(* Logix 5000 project; controller Drives_Line1 1756-L72 rev 20.13; software revision 20.04; part 3 of 21 *)
(* tags used below, declared in another part *)
   Entry_PosPv_Shear_Stitch : REAL;
   Entry_PosPv_Stitch_HOC : DINT;
   Entry_PosSp_AtStitch_EOC : DINT;
   Entry_PosSp_AtStitch_HOC : DINT;
   EOC_PosStitchStep : DINT;
   HOC_ToStitchStep : DINT;
   ons : BOOL[32];
   zEntry_Dist_Pinch_Shear : REAL;
   zEntry_Dist_ShearToStitch : REAL;
   zMaxSpdEntryNotSync : REAL;
   Bridle_01 : UDT_Bridle_3M;
   Bridle_01_FB_Diff : REAL;
   Bridle_01_FB_Update_Valid : BOOL;
   Bridle_01b_FBCounts_mm : REAL;
   Bridle_04 : UDT_Bridle_3M;
   Entry_Accu : UDT_Entry_Accu;
   EntryCmd : UDT_Commands_Zone;
   EntryConfig : UDT_Config_Zone;
   EntryCtrl : UDT_Control_Zone;
   EntryFdbks : UDT_Feedbacks_Zone;
   EntrySetpoints : UDT_Setpoints_Zone;
   EntryStat : UDT_Status_Zone;
   Exit_Accu : UDT_Exit_Accu;
   ExitCmd : UDT_Commands_Zone;
   ExitConfig : UDT_Config_Zone;
   ExitFdbks : UDT_Feedbacks_Zone;
   ExitSetpoints : UDT_Setpoints_Zone;
   ExitStat : UDT_Status_Zone;
   In_Commands : UDT_Commands;
   In_Config : UDT_Config;
   In_Setpoints : UDT_Setpoints;
   LineStat : UDT_Status_Line;
   Out_Feedbacks : UDT_Fdbks;
   Out_Status : UDT_Status;
   Pinchroll_2_FB_Difference : DINT;
   Pinchroll_2_FB_Update_Valid : BOOL;
   Pinchroll_2_FBCounts_mm : REAL;
   Pinchroll_3 : UDT_Pinchroll;
   TestConfig_Entry : UDT_Config_Zone;
   Unwinder_1 : UDT_Unwinder;
   Unwinder_2 : UDT_Unwinder;
   Winder : UDT_Winder;
   zConfigFromMaster : BOOL;
(* P01_Entry_Zone, continued *)

ROUTINE R04a_EOC_ToStitch   (* ladder *)
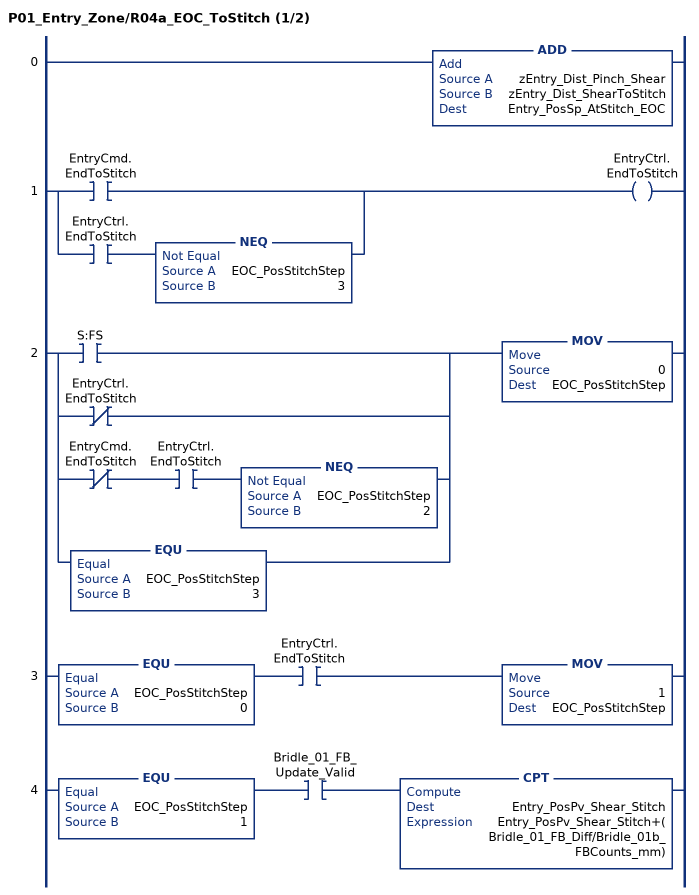
   0: ADD(zEntry_Dist_Pinch_Shear,zEntry_Dist_ShearToStitch,Entry_PosSp_AtStitch_EOC);
   1: [XIC(EntryCmd.EndToStitch) ,XIC(EntryCtrl.EndToStitch) NEQ(EOC_PosStitchStep,3) ]OTE(EntryCtrl.EndToStitch);
   2: [XIC(S:FS) ,XIO(EntryCtrl.EndToStitch) ,XIO(EntryCmd.EndToStitch) XIC(EntryCtrl.EndToStitch) NEQ(EOC_PosStitchStep,2) ,EQU(EOC_PosStitchStep,3) ]MOV(0,EOC_PosStitchStep);
   3: EQU(EOC_PosStitchStep,0)XIC(EntryCtrl.EndToStitch)MOV(1,EOC_PosStitchStep);
   4: EQU(EOC_PosStitchStep,1)XIC(Bridle_01_FB_Update_Valid)CPT(Entry_PosPv_Shear_Stitch,Entry_PosPv_Shear_Stitch+(Bridle_01_FB_Diff/Bridle_01b_FBCounts_mm));
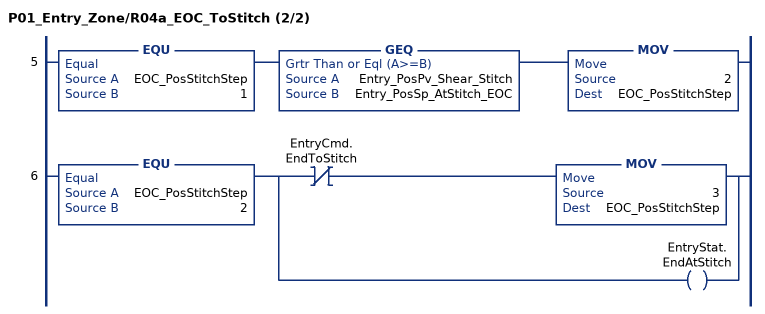
   5: EQU(EOC_PosStitchStep,1)GEQ(Entry_PosPv_Shear_Stitch,Entry_PosSp_AtStitch_EOC)MOV(2,EOC_PosStitchStep);
   6: EQU(EOC_PosStitchStep,2)[XIO(EntryCmd.EndToStitch) MOV(3,EOC_PosStitchStep) ,OTE(EntryStat.EndAtStitch) ];
END_ROUTINE

ROUTINE R04b_HOC_ToStitch   (* ladder *)
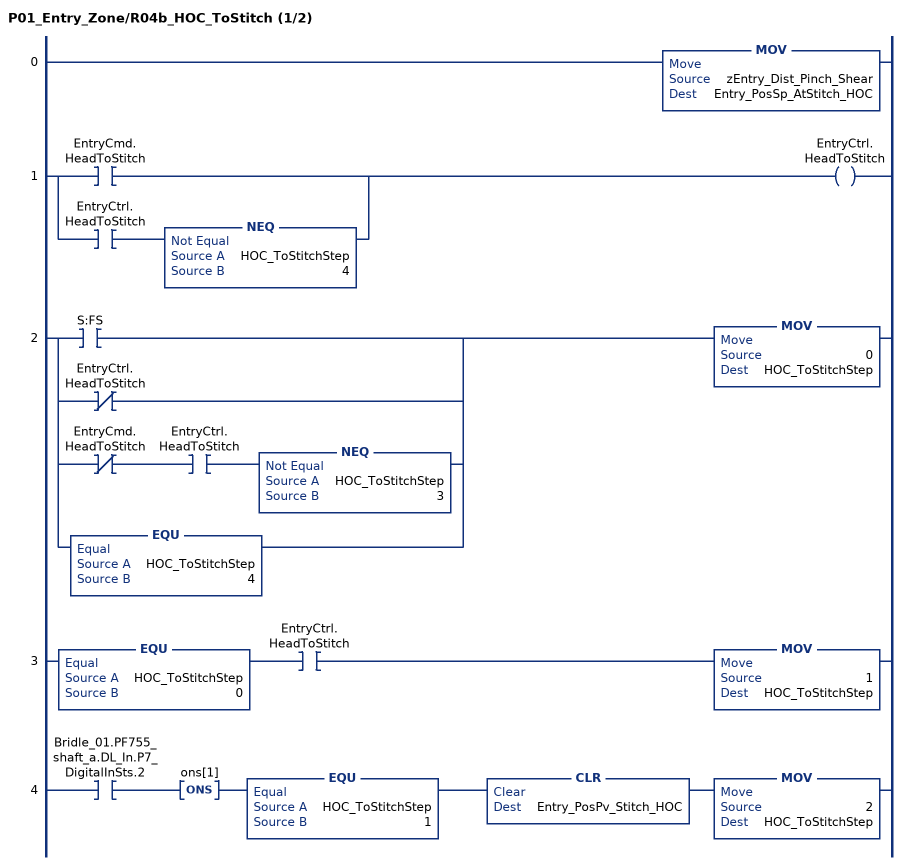
   0: MOV(zEntry_Dist_Pinch_Shear,Entry_PosSp_AtStitch_HOC);
   1: [XIC(EntryCmd.HeadToStitch) ,XIC(EntryCtrl.HeadToStitch) NEQ(HOC_ToStitchStep,4) ]OTE(EntryCtrl.HeadToStitch);
   2: [XIC(S:FS) ,XIO(EntryCtrl.HeadToStitch) ,XIO(EntryCmd.HeadToStitch) XIC(EntryCtrl.HeadToStitch) NEQ(HOC_ToStitchStep,3) ,EQU(HOC_ToStitchStep,4) ]MOV(0,HOC_ToStitchStep);
   3: EQU(HOC_ToStitchStep,0)XIC(EntryCtrl.HeadToStitch)MOV(1,HOC_ToStitchStep);
   4: XIC(Bridle_01.PF755_shaft_a.DL_In.P7_DigitalInSts.2)ONS(ons[1])EQU(HOC_ToStitchStep,1)CLR(Entry_PosPv_Stitch_HOC)MOV(2,HOC_ToStitchStep);
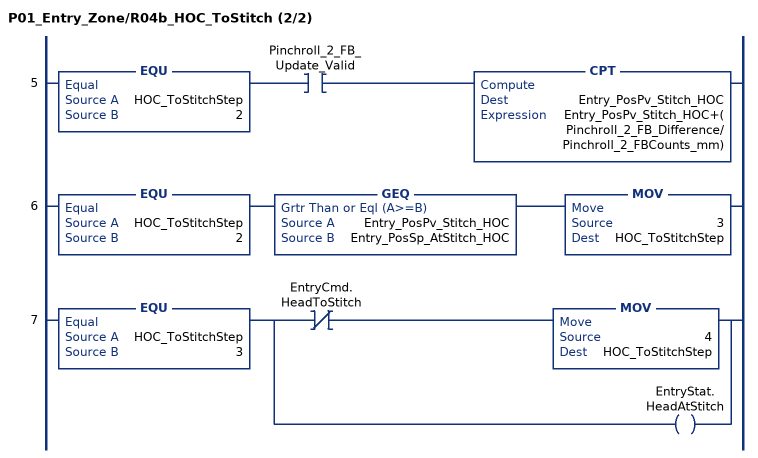
   5: EQU(HOC_ToStitchStep,2)XIC(Pinchroll_2_FB_Update_Valid)CPT(Entry_PosPv_Stitch_HOC,Entry_PosPv_Stitch_HOC+(Pinchroll_2_FB_Difference/Pinchroll_2_FBCounts_mm));
   6: EQU(HOC_ToStitchStep,2)GEQ(Entry_PosPv_Stitch_HOC,Entry_PosSp_AtStitch_HOC)MOV(3,HOC_ToStitchStep);
   7: EQU(HOC_ToStitchStep,3)[XIO(EntryCmd.HeadToStitch) MOV(4,HOC_ToStitchStep) ,OTE(EntryStat.HeadAtStitch) ];
END_ROUTINE

ROUTINE R06_Control   (* ladder *)
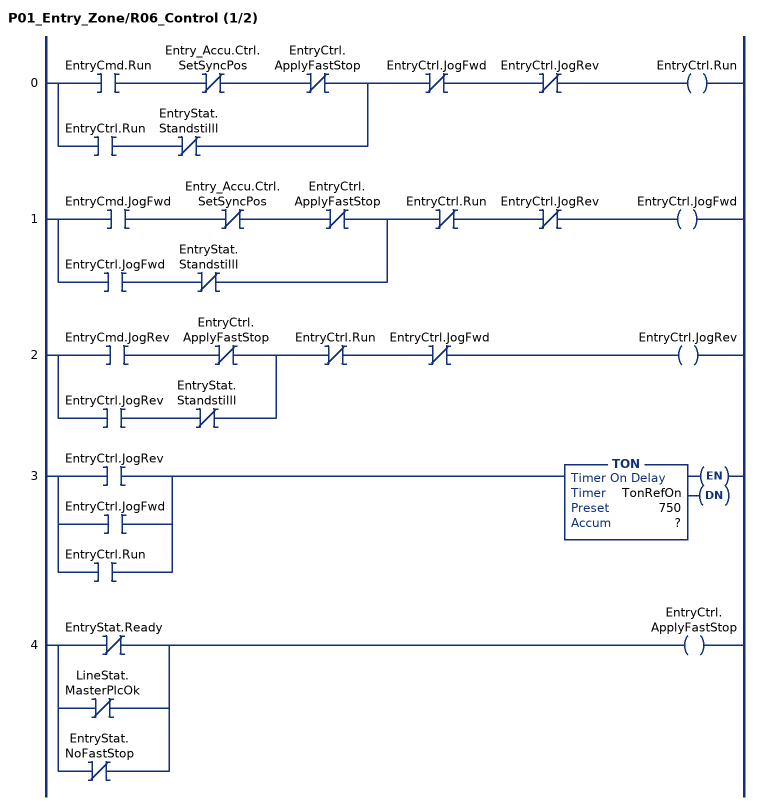
   0: [XIC(EntryCmd.Run) XIO(Entry_Accu.Ctrl.SetSyncPos) XIO(EntryCtrl.ApplyFastStop) ,XIC(EntryCtrl.Run) XIO(EntryStat.Standstilll) ]XIO(EntryCtrl.JogFwd)XIO(EntryCtrl.JogRev)OTE(EntryCtrl.Run);
   1: [XIC(EntryCmd.JogFwd) XIO(Entry_Accu.Ctrl.SetSyncPos) XIO(EntryCtrl.ApplyFastStop) ,XIC(EntryCtrl.JogFwd) XIO(EntryStat.Standstilll) ]XIO(EntryCtrl.Run)XIO(EntryCtrl.JogRev)OTE(EntryCtrl.JogFwd);
   2: [XIC(EntryCmd.JogRev) XIO(EntryCtrl.ApplyFastStop) ,XIC(EntryCtrl.JogRev) XIO(EntryStat.Standstilll) ]XIO(EntryCtrl.Run)XIO(EntryCtrl.JogFwd)OTE(EntryCtrl.JogRev);
   3: [XIC(EntryCtrl.JogRev) ,XIC(EntryCtrl.JogFwd) ,XIC(EntryCtrl.Run) ]TON(TonRefOn,?,?);
   4: [XIO(EntryStat.Ready) ,XIO(LineStat.MasterPlcOk) ,XIO(EntryStat.NoFastStop) ]OTE(EntryCtrl.ApplyFastStop);
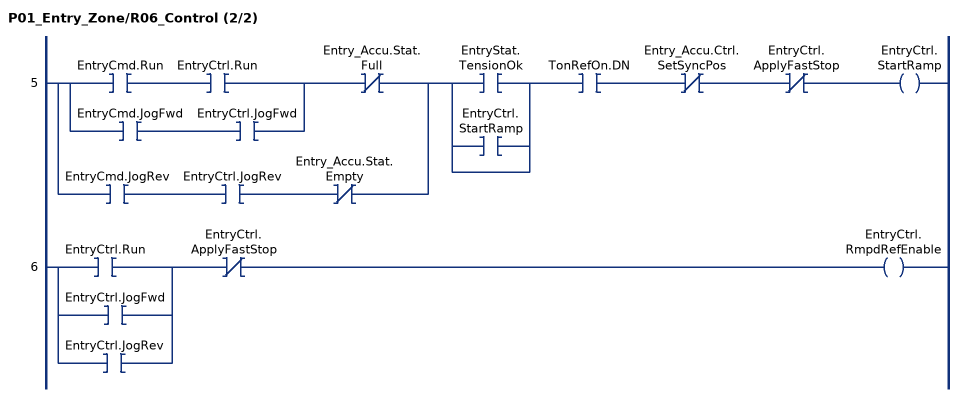
   5: [[XIC(EntryCmd.Run) XIC(EntryCtrl.Run) ,XIC(EntryCmd.JogFwd) XIC(EntryCtrl.JogFwd) ] XIO(Entry_Accu.Stat.Full) ,XIC(EntryCmd.JogRev) XIC(EntryCtrl.JogRev) XIO(Entry_Accu.Stat.Empty) ][XIC(EntryStat.TensionOk) ,XIC(EntryCtrl.StartRamp) ,]XIC(TonRefOn.DN)XIO(Entry_Accu.Ctrl.SetSyncPos)XIO(EntryCtrl.ApplyFastStop)OTE(EntryCtrl.StartRamp);
   6: [XIC(EntryCtrl.Run) ,XIC(EntryCtrl.JogFwd) ,XIC(EntryCtrl.JogRev) ]XIO(EntryCtrl.ApplyFastStop)OTE(EntryCtrl.RmpdRefEnable);
END_ROUTINE

ROUTINE R07_Ramp_EntryRef_Ve   (* function block diagram *)
   SHEET 1   // Limit speed reference
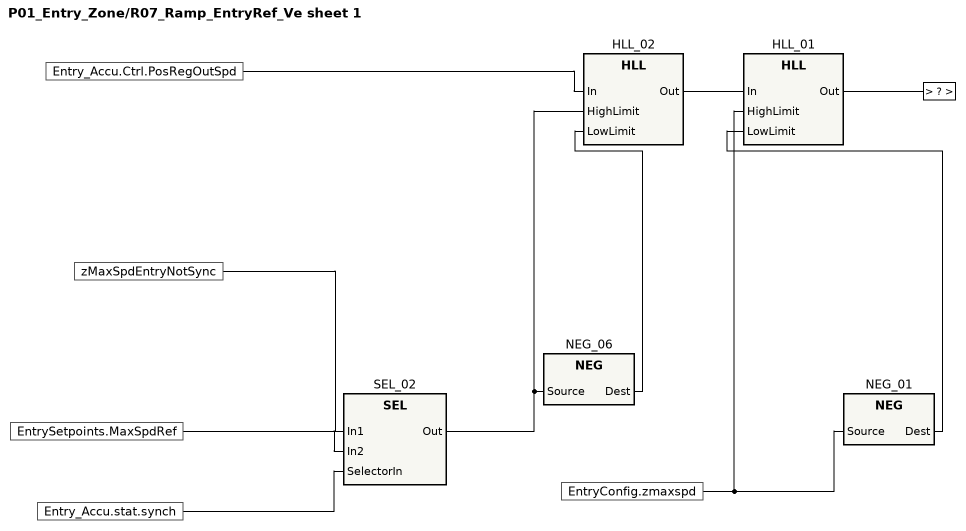
   SEL_02 : SEL(In1 := zMaxSpdEntryNotSync, In2 := EntrySetpoints.MaxSpdRef, SelectorIn := Entry_Accu.stat.synch);
   NEG_06 : NEG(Source := SEL_02.Out);
   HLL_02 : HLL(In := Entry_Accu.Ctrl.PosRegOutSpd, HighLimit := SEL_02.Out, LowLimit := NEG_06.Dest);
   NEG_01 : NEG(Source := EntryConfig.zmaxspd);
   HLL_01 : HLL(In := HLL_02.Out, HighLimit := EntryConfig.zmaxspd, LowLimit := NEG_01.Dest);
   WIRE(?) := HLL_01.Out;
   SHEET 2   // Select reference
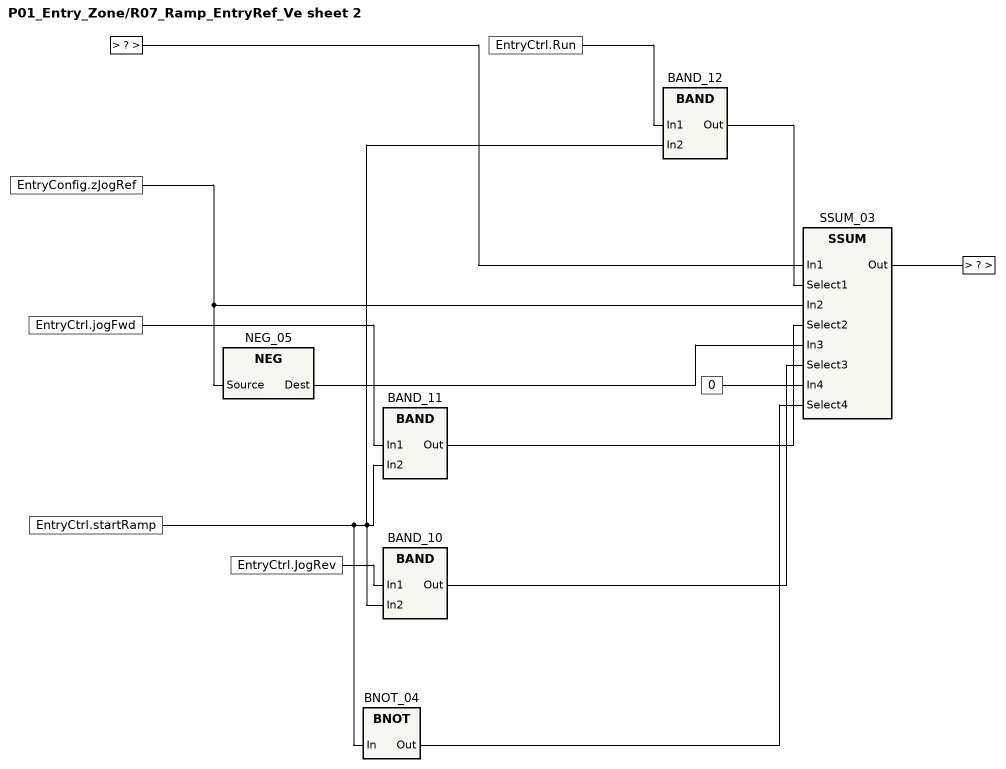
   NEG_05 : NEG(Source := EntryConfig.zJogRef);
   BNOT_04 : BNOT(In := EntryCtrl.startRamp);
   BAND_11 : BAND(In1 := EntryCtrl.jogFwd, In2 := EntryCtrl.startRamp);
   BAND_10 : BAND(In1 := EntryCtrl.JogRev, In2 := EntryCtrl.startRamp);
   BAND_12 : BAND(In1 := EntryCtrl.Run, In2 := EntryCtrl.startRamp);
   SSUM_03 : SSUM(In1 := WIRE(?), Select1 := BAND_12.Out, In2 := EntryConfig.zJogRef, Select2 := BAND_11.Out, In3 := NEG_05.Dest, Select3 := BAND_10.Out, In4 := 0, Select4 := BNOT_04.Out);
   WIRE(?) := SSUM_03.Out;
   SHEET 3   // Select acceleration rate
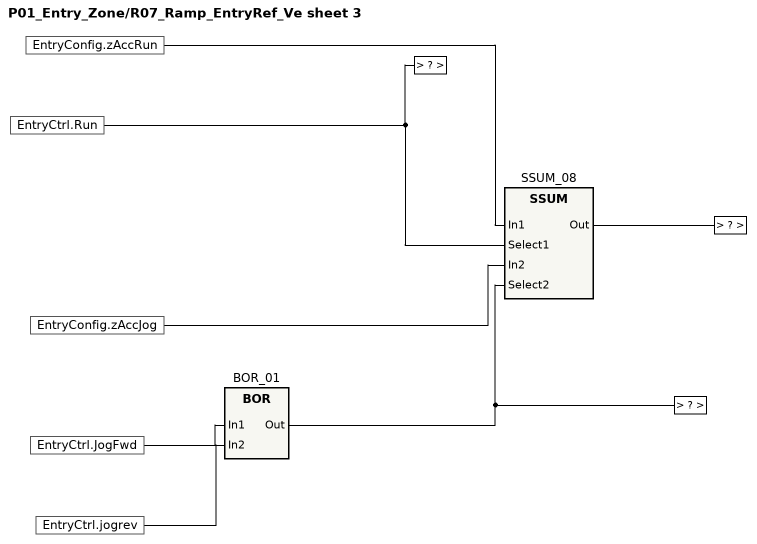
   BOR_01 : BOR(In1 := EntryCtrl.JogFwd, In2 := EntryCtrl.jogrev);
   WIRE(?) := EntryCtrl.Run;
   SSUM_08 : SSUM(In1 := EntryConfig.zAccRun, Select1 := EntryCtrl.Run, In2 := EntryConfig.zAccJog, Select2 := BOR_01.Out);
   WIRE(?) := BOR_01.Out;
   WIRE(?) := SSUM_08.Out;
   SHEET 4   // Select deceleration rate
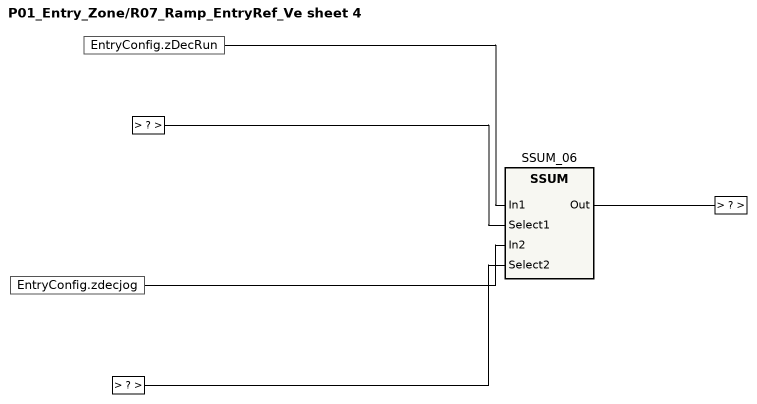
   SSUM_06 : SSUM(In1 := EntryConfig.zDecRun, Select1 := WIRE(?), In2 := EntryConfig.zdecjog, Select2 := WIRE(?));
   WIRE(?) := SSUM_06.Out;
   SHEET 5   // Select jerk rate
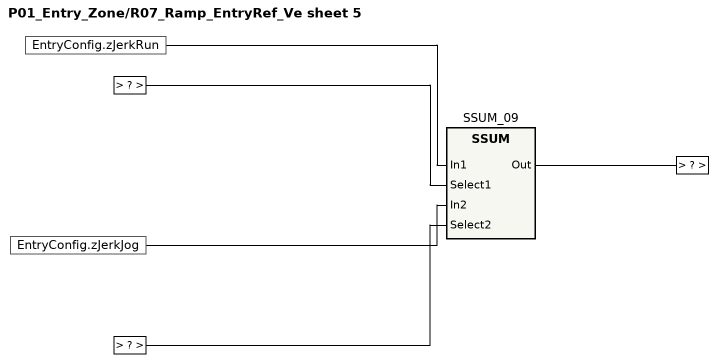
   SSUM_09 : SSUM(In1 := EntryConfig.zJerkRun, Select1 := WIRE(?), In2 := EntryConfig.zJerkJog, Select2 := WIRE(?));
   WIRE(?) := SSUM_09.Out;
   SHEET 6   // S-Curve entry speed (Ve)
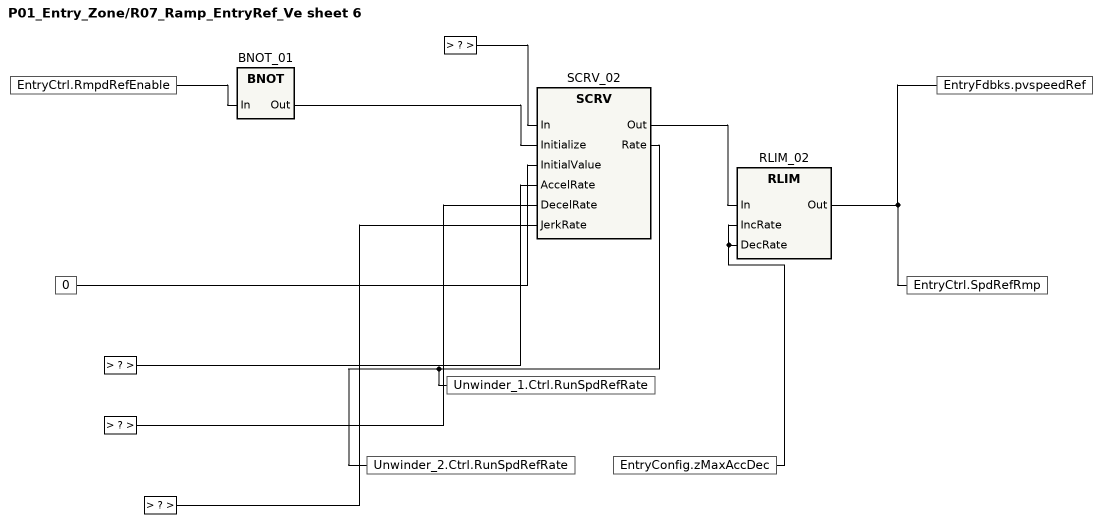
   BNOT_01 : BNOT(In := EntryCtrl.RmpdRefEnable);
   SCRV_02 : SCRV(In := WIRE(?), Initialize := BNOT_01.Out, InitialValue := 0, AccelRate := WIRE(?), DecelRate := WIRE(?), JerkRate := WIRE(?));
   Unwinder_2.Ctrl.RunSpdRefRate := SCRV_02.Rate;
   Unwinder_1.Ctrl.RunSpdRefRate := SCRV_02.Rate;
   RLIM_02 : RLIM(In := SCRV_02.Out, IncRate := EntryConfig.zMaxAccDec, DecRate := EntryConfig.zMaxAccDec);
   EntryCtrl.SpdRefRmp := RLIM_02.Out;
   EntryFdbks.pvspeedRef := RLIM_02.Out;
END_ROUTINE

ROUTINE R999_Test   (* ladder *)
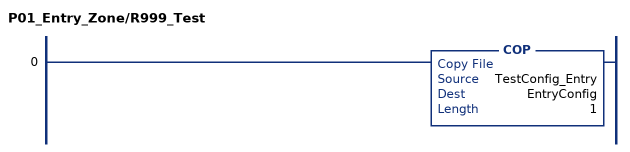
   0: COP(TestConfig_Entry,EntryConfig,1);
END_ROUTINE

ROUTINE R99_To_Master   (* ladder *)
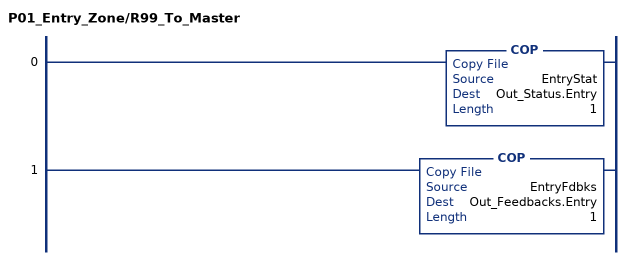
   0: COP(EntryStat,Out_Status.Entry,1);
   1: COP(EntryFdbks,Out_Feedbacks.Entry,1);
END_ROUTINE
END_PROGRAM

PROGRAM P02_Exit_Zone   (* main routine R00_Main *)
VAR
   BAND_10 : FBD_BOOLEAN_AND := (In3 := 1, In4 := 1, In5 := 1, In6 := 1, In7 := 1, In8 := 1);
   BAND_11 : FBD_BOOLEAN_AND := (In3 := 1, In4 := 1, In5 := 1, In6 := 1, In7 := 1, In8 := 1);
   BAND_12 : FBD_BOOLEAN_AND := (In3 := 1, In4 := 1, In5 := 1, In6 := 1, In7 := 1, In8 := 1);
   BNOT_02 : FBD_BOOLEAN_NOT := (Out := 1);
   BNOT_04 : FBD_BOOLEAN_NOT := (Out := 1);
   BOR_02 : FBD_BOOLEAN_OR;
   DIV_02 : FBD_MATH := (SourceA := 70.46141, SourceB := 100.0, Dest := 0.7046141);
   EOC_ToCoilerStep : DINT;
   Exit_PosPv_Winder : REAL;
   HLL_03 : HL_LIMIT := (HighAlarm := 1, LowAlarm := 1, Status := 16#0000_0003, InstructFault := 1, LimitsInv := 1);
   HLL_04 : HL_LIMIT := (HighLimit := 0.35230705, LowLimit := -0.35230705);
   MUL_02 : FBD_MATH := (SourceA := 0.5, SourceB := 0.7046141, Dest := 0.35230705);
   NEG_04 : FBD_MATH_ADVANCED := (Source := 0.35230705, Dest := -0.35230705);
   NEG_05 : FBD_MATH_ADVANCED := (Source := 0.116, Dest := -0.116);
   NEG_06 : FBD_MATH_ADVANCED;
   RLIM_03 : RATE_LIMITER := (IncRate := 0.25, DecRate := 0.25, RTSTime := 1, DeltaT := 0.05);
   SCL_02 : SCALE := (In := 709.3403, InRawMax := 1000.0, InRawMin := 508.0, InEUMax := 100.0, InEUMin := 50.0, Limiting := 1, Out := 70.46141);
   SCRV_03 : S_CURVE := (Initialize := 1, RTSTime := 1, DeltaT := 0.05);
   SEL_02 : SELECT := (In1 := 0.025, SelectorIn := 1);
   SSUM_03 : SELECTED_SUMMER := (Gain1 := 1.0, In2 := 0.116, Gain2 := 1.0, In3 := -0.116, Gain3 := 1.0, Gain4 := 1.0, Select4 := 1, Gain5 := 1.0, Gain6 := 1.0, Gain7 := 1.0, Gain8 := 1.0);
   SSUM_07 : SELECTED_SUMMER := (In1 := 0.04, Gain1 := 1.0, In2 := 0.083, Gain2 := 1.0, Gain3 := 1.0, Gain4 := 1.0, Gain5 := 1.0, Gain6 := 1.0, Gain7 := 1.0, Gain8 := 1.0);
   SSUM_10 : SELECTED_SUMMER := (In1 := 0.04, Gain1 := 1.0, In2 := 0.083, Gain2 := 1.0, Gain3 := 1.0, Gain4 := 1.0, Gain5 := 1.0, Gain6 := 1.0, Gain7 := 1.0, Gain8 := 1.0);
   SSUM_11 : SELECTED_SUMMER := (In1 := 0.15, Gain1 := 1.0, In2 := 0.25, Gain2 := 1.0, Gain3 := 1.0, Gain4 := 1.0, Gain5 := 1.0, Gain6 := 1.0, Gain7 := 1.0, Gain8 := 1.0);
   TonRefOn : TIMER := (PRE := 750);
   zMaxSpdExitNotSync : REAL := 0.025;
END_VAR

ROUTINE R00_Main   (* ladder *)
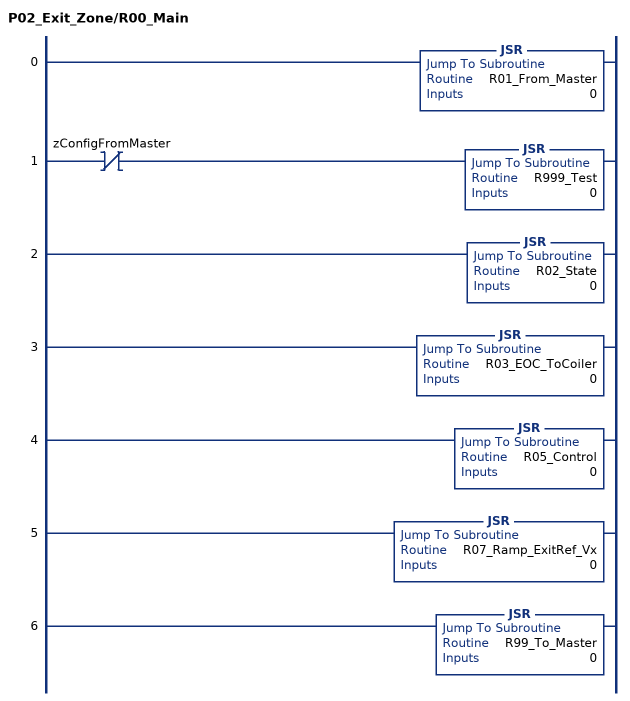
   0: JSR(R01_From_Master,0);
   1: XIO(zConfigFromMaster)JSR(R999_Test,0);
   2: JSR(R02_State,0);
   3: JSR(R03_EOC_ToCoiler,0);
   4: JSR(R05_Control,0);
   5: JSR(R07_Ramp_ExitRef_Vx,0);
   6: JSR(R99_To_Master,0);
END_ROUTINE

ROUTINE R01_From_Master   (* ladder *)
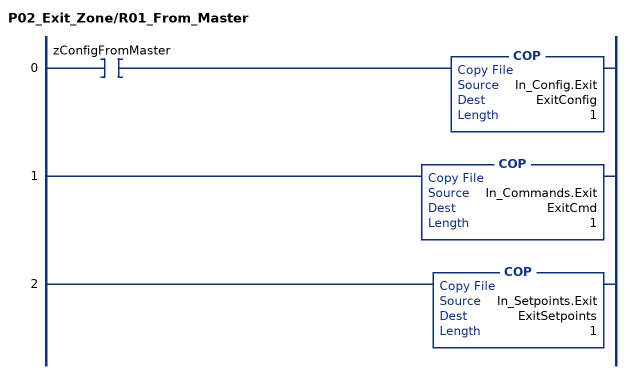
   0: XIC(zConfigFromMaster)COP(In_Config.Exit,ExitConfig,1);
   1: COP(In_Commands.Exit,ExitCmd,1);
   2: COP(In_Setpoints.Exit,ExitSetpoints,1);
END_ROUTINE

ROUTINE R02_State   (* ladder *)
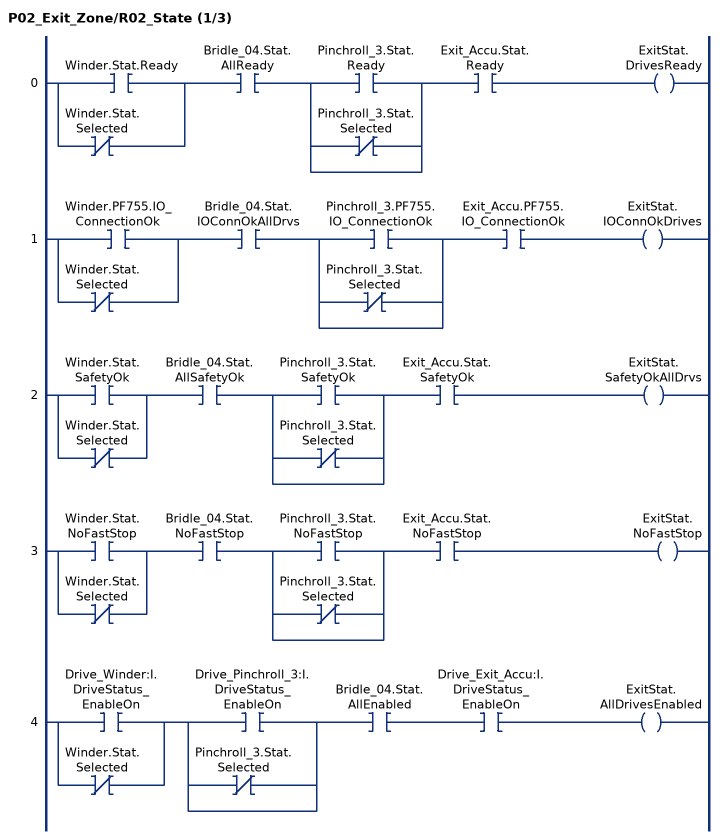
   0: [XIC(Winder.Stat.Ready) ,XIO(Winder.Stat.Selected) ]XIC(Bridle_04.Stat.AllReady)[XIC(Pinchroll_3.Stat.Ready) ,XIO(Pinchroll_3.Stat.Selected) ,]XIC(Exit_Accu.Stat.Ready)OTE(ExitStat.DrivesReady);
   1: [XIC(Winder.PF755.IO_ConnectionOk) ,XIO(Winder.Stat.Selected) ]XIC(Bridle_04.Stat.IOConnOkAllDrvs)[XIC(Pinchroll_3.PF755.IO_ConnectionOk) ,XIO(Pinchroll_3.Stat.Selected) ,]XIC(Exit_Accu.PF755.IO_ConnectionOk)OTE(ExitStat.IOConnOkDrives);
   2: [XIC(Winder.Stat.SafetyOk) ,XIO(Winder.Stat.Selected) ]XIC(Bridle_04.Stat.AllSafetyOk)[XIC(Pinchroll_3.Stat.SafetyOk) ,XIO(Pinchroll_3.Stat.Selected) ,]XIC(Exit_Accu.Stat.SafetyOk)OTE(ExitStat.SafetyOkAllDrvs);
   3: [XIC(Winder.Stat.NoFastStop) ,XIO(Winder.Stat.Selected) ]XIC(Bridle_04.Stat.NoFastStop)[XIC(Pinchroll_3.Stat.NoFastStop) ,XIO(Pinchroll_3.Stat.Selected) ,]XIC(Exit_Accu.Stat.NoFastStop)OTE(ExitStat.NoFastStop);
   4: [XIC(Drive_Winder:I.DriveStatus_EnableOn) ,XIO(Winder.Stat.Selected) ][XIC(Drive_Pinchroll_3:I.DriveStatus_EnableOn) ,XIO(Pinchroll_3.Stat.Selected) ,]XIC(Bridle_04.Stat.AllEnabled)XIC(Drive_Exit_Accu:I.DriveStatus_EnableOn)OTE(ExitStat.AllDrivesEnabled);
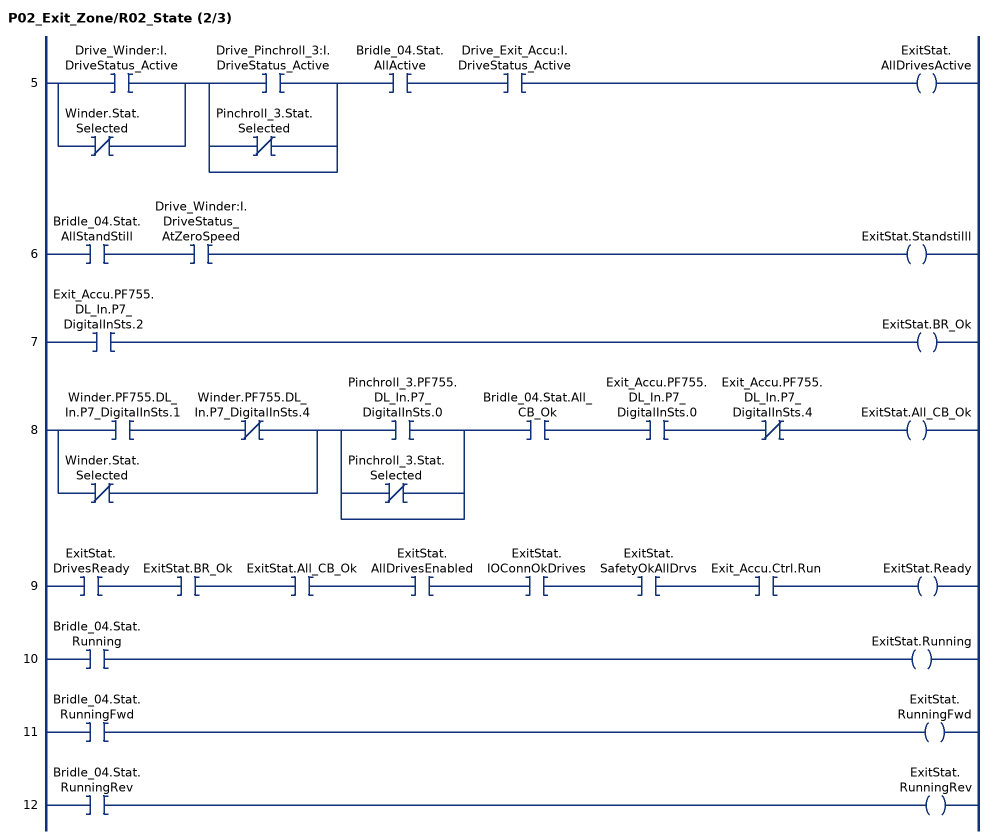
   5: [XIC(Drive_Winder:I.DriveStatus_Active) ,XIO(Winder.Stat.Selected) ][XIC(Drive_Pinchroll_3:I.DriveStatus_Active) ,XIO(Pinchroll_3.Stat.Selected) ,]XIC(Bridle_04.Stat.AllActive)XIC(Drive_Exit_Accu:I.DriveStatus_Active)OTE(ExitStat.AllDrivesActive);
   6: XIC(Bridle_04.Stat.AllStandStill)XIC(Drive_Winder:I.DriveStatus_AtZeroSpeed)OTE(ExitStat.Standstilll);
   7: XIC(Exit_Accu.PF755.DL_In.P7_DigitalInSts.2)OTE(ExitStat.BR_Ok);
   8: [XIC(Winder.PF755.DL_In.P7_DigitalInSts.1) XIO(Winder.PF755.DL_In.P7_DigitalInSts.4) ,XIO(Winder.Stat.Selected) ][XIC(Pinchroll_3.PF755.DL_In.P7_DigitalInSts.0) ,XIO(Pinchroll_3.Stat.Selected) ,]XIC(Bridle_04.Stat.All_CB_Ok)XIC(Exit_Accu.PF755.DL_In.P7_DigitalInSts.0)XIO(Exit_Accu.PF755.DL_In.P7_DigitalInSts.4)OTE(ExitStat.All_CB_Ok);
   9: XIC(ExitStat.DrivesReady)XIC(ExitStat.BR_Ok)XIC(ExitStat.All_CB_Ok)XIC(ExitStat.AllDrivesEnabled)XIC(ExitStat.IOConnOkDrives)XIC(ExitStat.SafetyOkAllDrvs)XIC(Exit_Accu.Ctrl.Run)OTE(ExitStat.Ready);
   10: XIC(Bridle_04.Stat.Running)OTE(ExitStat.Running);
   11: XIC(Bridle_04.Stat.RunningFwd)OTE(ExitStat.RunningFwd);
   12: XIC(Bridle_04.Stat.RunningRev)OTE(ExitStat.RunningRev);
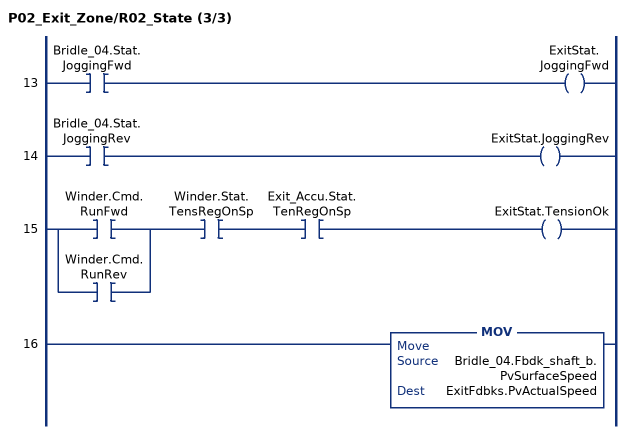
   13: XIC(Bridle_04.Stat.JoggingFwd)OTE(ExitStat.JoggingFwd);
   14: XIC(Bridle_04.Stat.JoggingRev)OTE(ExitStat.JoggingRev);
   15: [XIC(Winder.Cmd.RunFwd) ,XIC(Winder.Cmd.RunRev) ]XIC(Winder.Stat.TensRegOnSp)XIC(Exit_Accu.Stat.TenRegOnSp)OTE(ExitStat.TensionOk);
   16: MOV(Bridle_04.Fbdk_shaft_b.PvSurfaceSpeed,ExitFdbks.PvActualSpeed);
END_ROUTINE
